FUNCTION ASSEMBLE_WORD_FROM_BOOLS (* this Function combines the 16 BOOLS to a WORD *)
  (* Standard: 61499-1; Description: Copyright (c) 2024 HR Agrartechnik GmbH This program and the accompanying materials are made available under the terms of the Eclipse Public License 2.0 which is available at https://www.eclipse.org/legal/epl-2.0/ SPDX-License-Identifier: EPL-2.0 *)
  (* Version 1.0, 2024-02-22, Franz Höpfinger, HR Agrartechnik, initial Implementation *)
  (* Version 1.1, 2024-07-28, Moritz Ortmeier, HR Agrartechnik, rename Function and change Input/Output Variables *)
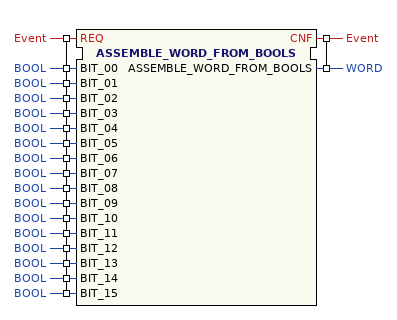
  EVENT_INPUT
    REQ WITH BIT_00, BIT_01, BIT_02, BIT_03, BIT_04, BIT_05, BIT_06, BIT_07, BIT_08, BIT_09, BIT_10, BIT_11, BIT_12, BIT_13, BIT_14, BIT_15;
  END_EVENT
  EVENT_OUTPUT
    CNF WITH ASSEMBLE_WORD_FROM_BOOLS;
  END_EVENT
  VAR_INPUT
    BIT_00 : BOOL;
    BIT_01 : BOOL;
    BIT_02 : BOOL;
    BIT_03 : BOOL;
    BIT_04 : BOOL;
    BIT_05 : BOOL;
    BIT_06 : BOOL;
    BIT_07 : BOOL;
    BIT_08 : BOOL;
    BIT_09 : BOOL;
    BIT_10 : BOOL;
    BIT_11 : BOOL;
    BIT_12 : BOOL;
    BIT_13 : BOOL;
    BIT_14 : BOOL;
    BIT_15 : BOOL;
  END_VAR
  VAR_OUTPUT
    ASSEMBLE_WORD_FROM_BOOLS : WORD;
  END_VAR
  BODY IN ST:
(* this Function combines the 16 BOOLS to a WORD *)
FUNCTION ASSEMBLE_WORD_FROM_BOOLS : WORD

VAR_INPUT
	BIT_00 : BOOL;
	BIT_01 : BOOL;
	BIT_02 : BOOL;
	BIT_03 : BOOL;
	BIT_04 : BOOL;
	BIT_05 : BOOL;
	BIT_06 : BOOL;
	BIT_07 : BOOL;
	BIT_08 : BOOL;
	BIT_09 : BOOL;
	BIT_10 : BOOL;
	BIT_11 : BOOL;
	BIT_12 : BOOL;
	BIT_13 : BOOL;
	BIT_14 : BOOL;
	BIT_15 : BOOL;
END_VAR

ASSEMBLE_WORD_FROM_BOOLS.%X0 := BIT_00;
ASSEMBLE_WORD_FROM_BOOLS.%X1 := BIT_01;
ASSEMBLE_WORD_FROM_BOOLS.%X2 := BIT_02;
ASSEMBLE_WORD_FROM_BOOLS.%X3 := BIT_03;
ASSEMBLE_WORD_FROM_BOOLS.%X4 := BIT_04;
ASSEMBLE_WORD_FROM_BOOLS.%X5 := BIT_05;
ASSEMBLE_WORD_FROM_BOOLS.%X6 := BIT_06;
ASSEMBLE_WORD_FROM_BOOLS.%X7 := BIT_07;
ASSEMBLE_WORD_FROM_BOOLS.%X8 := BIT_08;
ASSEMBLE_WORD_FROM_BOOLS.%X9 := BIT_09;
ASSEMBLE_WORD_FROM_BOOLS.%X10 := BIT_10;
ASSEMBLE_WORD_FROM_BOOLS.%X11 := BIT_11;
ASSEMBLE_WORD_FROM_BOOLS.%X12 := BIT_12;
ASSEMBLE_WORD_FROM_BOOLS.%X13 := BIT_13;
ASSEMBLE_WORD_FROM_BOOLS.%X14 := BIT_14;
ASSEMBLE_WORD_FROM_BOOLS.%X15 := BIT_15;

END_FUNCTION
  END_BODY
END_FUNCTION
